TYPE ST_ItemSimulator_HMI_Status :
STRUCT
END_STRUCT
END_TYPE

(* stored: Version 1.1.0.1, ProductVersion 3.1.4024.12
   DUT ST_ItemSimulator_HMI_Status: Id {fbdc06a8-5a54-40ca-a94c-e0eb3cdf61ed} *)
